TYPE DUT_HMI_Valve EXTENDS DUT_Com_Base_Valve :
STRUCT
	ModeValue : INT:= 1; // 0: Manual; 1: Auto;
	DisableAutoManual : BOOL;
END_STRUCT
END_TYPE

(* stored: Version 1.1.0.1, ProductVersion 3.1.4024.12
   DUT DUT_HMI_Valve: Id {7e2b4294-76ca-47d6-8c7b-fda0034aae6c} *)
